ABB RAPID module: Module1.mod

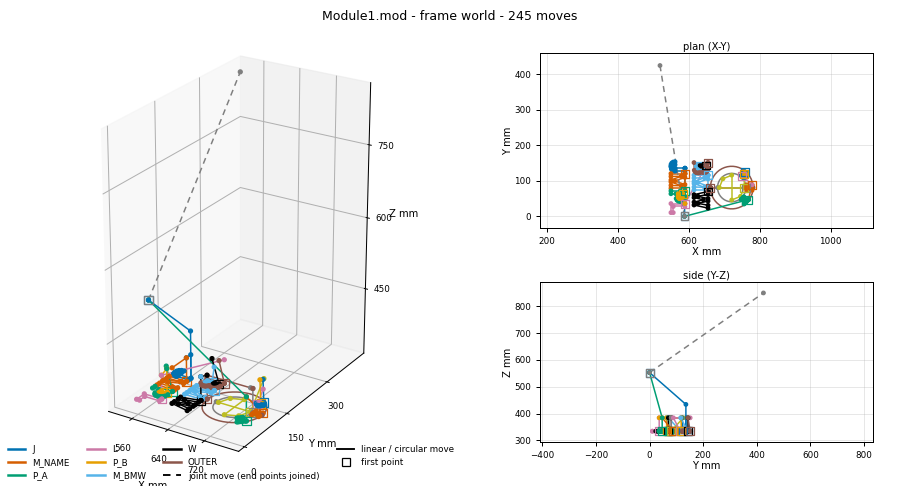
[picture p0: tool path of Module1.mod in frame world, 245 of 245 moves have a stored position in this frame; points joined in program order, loops and branches not executed]
MODULE Module1
    TASK PERS tooldata TCP_JMPL:=[TRUE,[[0,0,0],[1,0,0,0]],[1,[0,0,1],[1,0,0,0],0,0,0]];
    TASK PERS wobjdata WOB_LAB1:=[FALSE,TRUE,"",[[787.383,-61.438566881,334.26555336],[0.707106781,0,0,0.707106781]],[[0,0,0],[1,0,0,0]]];
    CONST robtarget J_10:=[[197.01,198.002626654,0.000000056],[-0.000000001,0.707106782,0.707106781,0],[0,0,0,0],[9E+09,9E+09,9E+09,9E+09,9E+09,9E+09]];
    CONST robtarget J_20:=[[197.01,225.346445883,0.000000064],[-0.000000001,0.707106782,0.707106781,0],[0,0,0,0],[9E+09,9E+09,9E+09,9E+09,9E+09,9E+09]];
    CONST robtarget J_30:=[[198.394,229.904456194,0.000000065],[-0.000000001,0.707106782,0.707106781,0],[0,0,0,0],[9E+09,9E+09,9E+09,9E+09,9E+09,9E+09]];
    CONST robtarget J_40:=[[202.114,231.501103306,0.000000066],[-0.000000001,0.707106782,0.707106781,0],[0,0,0,0],[9E+09,9E+09,9E+09,9E+09,9E+09,9E+09]];
    CONST robtarget J_50:=[[205.964,230.120830869,0.000000065],[-0.000000001,0.707106782,0.707106781,0],[0,0,0,0],[9E+09,9E+09,9E+09,9E+09,9E+09,9E+09]];
    CONST robtarget J_60:=[[206.878,228.358720771,0.000000065],[-0.000000001,0.707106782,0.707106781,0],[0,0,0,0],[9E+09,9E+09,9E+09,9E+09,9E+09,9E+09]];
    CONST robtarget J_70:=[[207.183,225.832935348,0.000000064],[-0.000000001,0.707106782,0.707106781,0],[0,0,0,0],[9E+09,9E+09,9E+09,9E+09,9E+09,9E+09]];
    CONST robtarget J_80:=[[215.378,225.832935348,0.000000064],[-0.000000001,0.707106782,0.707106781,0],[0,0,0,0],[9E+09,9E+09,9E+09,9E+09,9E+09,9E+09]];
    CONST robtarget J_90:=[[214.503,231.006128559,0.000000065],[-0.000000001,0.707106782,0.707106781,0],[0,0,0,0],[9E+09,9E+09,9E+09,9E+09,9E+09,9E+09]];
    CONST robtarget J_100:=[[211.879,234.85703209,0.000000067],[-0.000000001,0.707106782,0.707106781,0],[0,0,0,0],[9E+09,9E+09,9E+09,9E+09,9E+09,9E+09]];
    CONST robtarget J_110:=[[207.689,237.248467224,0.000000067],[-0.000000001,0.707106782,0.707106781,0],[0,0,0,0],[9E+09,9E+09,9E+09,9E+09,9E+09,9E+09]];
    CONST robtarget J_120:=[[202.114,238.046083673,0.000000067],[-0.000000001,0.707106782,0.707106781,0],[0,0,0,0],[9E+09,9E+09,9E+09,9E+09,9E+09,9E+09]];
    CONST robtarget J_130:=[[195.247,236.470649764,0.000000067],[-0.000000001,0.707106782,0.707106781,0],[0,0,0,0],[9E+09,9E+09,9E+09,9E+09,9E+09,9E+09]];
    CONST robtarget J_140:=[[192.552,234.567118309,0.000000066],[-0.000000001,0.707106782,0.707106781,0],[0,0,0,0],[9E+09,9E+09,9E+09,9E+09,9E+09,9E+09]];
    CONST robtarget J_150:=[[189.293,228.894707711,0.000000065],[-0.000000001,0.707106782,0.707106781,0],[0,0,0,0],[9E+09,9E+09,9E+09,9E+09,9E+09,9E+09]];
    CONST robtarget J_160:=[[188.876,225.346445883,0.000000064],[-0.000000001,0.707106782,0.707106781,0],[0,0,0,0],[9E+09,9E+09,9E+09,9E+09,9E+09,9E+09]];
    CONST robtarget J_170:=[[188.876,198.002626654,0.000000056],[-0.000000001,0.707106782,0.707106781,0],[0,0,0,0],[9E+09,9E+09,9E+09,9E+09,9E+09,9E+09]];
    CONST robtarget J_180:=[[197.01,198.002626654,0.000000056],[-0.000000001,0.707106782,0.707106781,0],[0,0,0,0],[9E+09,9E+09,9E+09,9E+09,9E+09,9E+09]];
    CONST robtarget M_NAME_10:=[[181.905,198.002626654,0.000000056],[-0.000000001,0.707106782,0.707106781,0],[0,0,0,0],[9E+09,9E+09,9E+09,9E+09,9E+09,9E+09]];
    CONST robtarget M_NAME_20:=[[181.905,237.500197238,0.000000067],[-0.000000001,0.707106782,0.707106781,0],[0,0,0,0],[9E+09,9E+09,9E+09,9E+09,9E+09,9E+09]];
    CONST robtarget M_NAME_30:=[[173.763,237.500197238,0.000000067],[-0.000000001,0.707106782,0.707106781,0],[0,0,0,0],[9E+09,9E+09,9E+09,9E+09,9E+09,9E+09]];
    CONST robtarget M_NAME_40:=[[174.579,208.090211995,0.000000059],[-0.000000001,0.707106782,0.707106781,0],[0,0,0,0],[9E+09,9E+09,9E+09,9E+09,9E+09,9E+09]];
    CONST robtarget M_NAME_50:=[[163.945,237.500197238,0.000000067],[-0.000000001,0.707106782,0.707106781,0],[0,0,0,0],[9E+09,9E+09,9E+09,9E+09,9E+09,9E+09]];
    CONST robtarget M_NAME_60:=[[158.355,237.500197238,0.000000067],[-0.000000001,0.707106782,0.707106781,0],[0,0,0,0],[9E+09,9E+09,9E+09,9E+09,9E+09,9E+09]];
    CONST robtarget M_NAME_70:=[[147.695,208.063341937,0.000000059],[-0.000000001,0.707106782,0.707106781,0],[0,0,0,0],[9E+09,9E+09,9E+09,9E+09,9E+09,9E+09]];
    CONST robtarget M_NAME_80:=[[148.511,237.500197238,0.000000067],[-0.000000001,0.707106782,0.707106781,0],[0,0,0,0],[9E+09,9E+09,9E+09,9E+09,9E+09,9E+09]];
    CONST robtarget M_NAME_90:=[[140.343,237.500197238,0.000000067],[-0.000000001,0.707106782,0.707106781,0],[0,0,0,0],[9E+09,9E+09,9E+09,9E+09,9E+09,9E+09]];
    CONST robtarget M_NAME_100:=[[140.343,198.002626654,0.000000056],[-0.000000001,0.707106782,0.707106781,0],[0,0,0,0],[9E+09,9E+09,9E+09,9E+09,9E+09,9E+09]];
    CONST robtarget M_NAME_110:=[[151.029,198.002626654,0.000000056],[-0.000000001,0.707106782,0.707106781,0],[0,0,0,0],[9E+09,9E+09,9E+09,9E+09,9E+09,9E+09]];
    CONST robtarget M_NAME_120:=[[161.124,226.648936574,0.000000064],[-0.000000001,0.707106782,0.707106781,0],[0,0,0,0],[9E+09,9E+09,9E+09,9E+09,9E+09,9E+09]];
    CONST robtarget M_NAME_130:=[[171.272,198.002626654,0.000000056],[-0.000000001,0.707106782,0.707106781,0],[0,0,0,0],[9E+09,9E+09,9E+09,9E+09,9E+09,9E+09]];
    CONST robtarget M_NAME_140:=[[181.905,198.002626654,0.000000056],[-0.000000001,0.707106782,0.707106781,0],[0,0,0,0],[9E+09,9E+09,9E+09,9E+09,9E+09,9E+09]];
    CONST robtarget P_A_10:=[[133.242,198.002626654,0.000000056],[-0.000000001,0.707106782,0.707106781,0],[0,0,0,0],[9E+09,9E+09,9E+09,9E+09,9E+09,9E+09]];
    CONST robtarget P_A_20:=[[133.242,237.500197238,0.000000067],[-0.000000001,0.707106782,0.707106781,0],[0,0,0,0],[9E+09,9E+09,9E+09,9E+09,9E+09,9E+09]];
    CONST robtarget P_A_30:=[[125.1,237.500197238,0.000000067],[-0.000000001,0.707106782,0.707106781,0],[0,0,0,0],[9E+09,9E+09,9E+09,9E+09,9E+09,9E+09]];
    CONST robtarget P_A_40:=[[125.1,223.584335784,0.000000063],[-0.000000001,0.707106782,0.707106781,0],[0,0,0,0],[9E+09,9E+09,9E+09,9E+09,9E+09,9E+09]];
    CONST robtarget P_A_50:=[[111.704,222.747121355,0.000000063],[-0.000000001,0.707106782,0.707106781,0],[0,0,0,0],[9E+09,9E+09,9E+09,9E+09,9E+09,9E+09]];
    CONST robtarget P_A_60:=[[106.966,220.234063855,0.000000062],[-0.000000001,0.707106782,0.707106781,0],[0,0,0,0],[9E+09,9E+09,9E+09,9E+09,9E+09,9E+09]];
    CONST robtarget P_A_70:=[[103.984,216.268609026,0.000000061],[-0.000000001,0.707106782,0.707106781,0],[0,0,0,0],[9E+09,9E+09,9E+09,9E+09,9E+09,9E+09]];
    CONST robtarget P_A_80:=[[102.99,211.075616825,0.00000006],[-0.000000001,0.707106782,0.707106781,0],[0,0,0,0],[9E+09,9E+09,9E+09,9E+09,9E+09,9E+09]];
    CONST robtarget P_A_90:=[[103.445,207.462301173,0.000000059],[-0.000000001,0.707106782,0.707106781,0],[0,0,0,0],[9E+09,9E+09,9E+09,9E+09,9E+09,9E+09]];
    CONST robtarget P_A_100:=[[104.809,204.257693241,0.000000058],[-0.000000001,0.707106782,0.707106781,0],[0,0,0,0],[9E+09,9E+09,9E+09,9E+09,9E+09,9E+09]];
    CONST robtarget P_A_110:=[[107.017,201.601800171,0.000000057],[-0.000000001,0.707106782,0.707106781,0],[0,0,0,0],[9E+09,9E+09,9E+09,9E+09,9E+09,9E+09]];
    CONST robtarget P_A_120:=[[110.004,199.630386465,0.000000057],[-0.000000001,0.707106782,0.707106781,0],[0,0,0,0],[9E+09,9E+09,9E+09,9E+09,9E+09,9E+09]];
    CONST robtarget P_A_130:=[[117.834,198.002626654,0.000000056],[-0.000000001,0.707106782,0.707106781,0],[0,0,0,0],[9E+09,9E+09,9E+09,9E+09,9E+09,9E+09]];
    CONST robtarget P_A_140:=[[133.242,198.002626654,0.000000056],[-0.000000001,0.707106782,0.707106781,0],[0,0,0,0],[9E+09,9E+09,9E+09,9E+09,9E+09,9E+09]];
    CONST robtarget L_10:=[[97.409,198.002626654,0.000000056],[-0.000000001,0.707106782,0.707106781,0],[0,-2,1,0],[9E+09,9E+09,9E+09,9E+09,9E+09,9E+09]];
    CONST robtarget L_20:=[[97.409,237.500197238,0.000000067],[-0.000000001,0.707106782,0.707106781,0],[0,-2,1,0],[9E+09,9E+09,9E+09,9E+09,9E+09,9E+09]];
    CONST robtarget L_30:=[[71.992,237.500197238,0.000000067],[-0.000000001,0.707106782,0.707106781,0],[0,-2,1,0],[9E+09,9E+09,9E+09,9E+09,9E+09,9E+09]];
    CONST robtarget L_40:=[[71.992,230.963702153,0.000000065],[-0.000000001,0.707106782,0.707106781,0],[0,-2,1,0],[9E+09,9E+09,9E+09,9E+09,9E+09,9E+09]];
    CONST robtarget L_50:=[[89.266,230.963702153,0.000000065],[-0.000000001,0.707106782,0.707106781,0],[0,-2,1,0],[9E+09,9E+09,9E+09,9E+09,9E+09,9E+09]];
    CONST robtarget L_60:=[[89.266,198.002626654,0.000000056],[-0.000000001,0.707106782,0.707106781,0],[0,-2,1,0],[9E+09,9E+09,9E+09,9E+09,9E+09,9E+09]];
    CONST robtarget L_70:=[[97.409,198.002626654,0.000000056],[-0.000000001,0.707106782,0.707106781,0],[0,-2,1,0],[9E+09,9E+09,9E+09,9E+09,9E+09,9E+09]];
    CONST robtarget P_B_100:=[[125.1,204.591447641,0.000000058],[-0.000000001,0.707106782,0.707106781,0],[0,0,0,0],[9E+09,9E+09,9E+09,9E+09,9E+09,9E+09]];
    CONST robtarget P_B_10:=[[125.1,204.591447641,0.000000058],[-0.000000001,0.707106782,0.707106781,0],[0,0,0,0],[9E+09,9E+09,9E+09,9E+09,9E+09,9E+09]];
    CONST robtarget P_B_20:=[[125.1,216.987029516,0.000000061],[-0.000000001,0.707106782,0.707106781,0],[0,0,0,0],[9E+09,9E+09,9E+09,9E+09,9E+09,9E+09]];
    CONST robtarget P_B_30:=[[117.834,216.987029516,0.000000061],[-0.000000001,0.707106782,0.707106781,0],[0,0,0,0],[9E+09,9E+09,9E+09,9E+09,9E+09,9E+09]];
    CONST robtarget P_B_40:=[[114.988,216.608020281,0.000000061],[-0.000000001,0.707106782,0.707106781,0],[0,0,0,0],[9E+09,9E+09,9E+09,9E+09,9E+09,9E+09]];
    CONST robtarget P_B_50:=[[112.908,215.46816415,0.000000061],[-0.000000001,0.707106782,0.707106781,0],[0,0,0,0],[9E+09,9E+09,9E+09,9E+09,9E+09,9E+09]];
    CONST robtarget P_B_60:=[[111.635,213.624029664,0.000000061],[-0.000000001,0.707106782,0.707106781,0],[0,0,0,0],[9E+09,9E+09,9E+09,9E+09,9E+09,9E+09]];
    CONST robtarget P_B_70:=[[111.211,211.127942727,0.00000006],[-0.000000001,0.707106782,0.707106781,0],[0,0,0,0],[9E+09,9E+09,9E+09,9E+09,9E+09,9E+09]];
    CONST robtarget P_B_80:=[[111.638,208.505990782,0.000000059],[-0.000000001,0.707106782,0.707106781,0],[0,0,0,0],[9E+09,9E+09,9E+09,9E+09,9E+09,9E+09]];
    CONST robtarget P_B_90:=[[114.957,205.083593961,0.000000058],[-0.000000001,0.707106782,0.707106781,0],[0,0,0,0],[9E+09,9E+09,9E+09,9E+09,9E+09,9E+09]];
    CONST robtarget P_B_110:=[[125.1,204.591447641,0.000000058],[-0.000000001,0.707106782,0.707106781,0],[0,0,0,0],[9E+09,9E+09,9E+09,9E+09,9E+09,9E+09]];
    CONST robtarget M_NAME_140_2:=[[177.487,133.0025429,0.000000038],[-0.000000001,0.707106782,0.707106781,0],[0,0,0,0],[9E+09,9E+09,9E+09,9E+09,9E+09,9E+09]];
    CONST robtarget M_NAME_10_2:=[[177.487,133.0025429,0.000000038],[-0.000000001,0.707106782,0.707106781,0],[0,0,0,0],[9E+09,9E+09,9E+09,9E+09,9E+09,9E+09]];
    CONST robtarget M_NAME_20_2:=[[177.487,172.500113484,0.000000049],[-0.000000001,0.707106782,0.707106781,0],[0,0,0,0],[9E+09,9E+09,9E+09,9E+09,9E+09,9E+09]];
    CONST robtarget M_NAME_30_2:=[[169.345,172.500113484,0.000000049],[-0.000000001,0.707106782,0.707106781,0],[0,0,0,0],[9E+09,9E+09,9E+09,9E+09,9E+09,9E+09]];
    CONST robtarget M_NAME_40_2:=[[170.161,143.090128241,0.000000041],[-0.000000001,0.707106782,0.707106781,0],[0,0,0,0],[9E+09,9E+09,9E+09,9E+09,9E+09,9E+09]];
    CONST robtarget M_NAME_50_2:=[[159.527,172.500113484,0.000000049],[-0.000000001,0.707106782,0.707106781,0],[0,0,0,0],[9E+09,9E+09,9E+09,9E+09,9E+09,9E+09]];
    CONST robtarget M_NAME_60_2:=[[153.937,172.500113484,0.000000049],[-0.000000001,0.707106782,0.707106781,0],[0,0,0,0],[9E+09,9E+09,9E+09,9E+09,9E+09,9E+09]];
    CONST robtarget M_NAME_70_2:=[[143.277,143.063258183,0.000000041],[-0.000000001,0.707106782,0.707106781,0],[0,0,0,0],[9E+09,9E+09,9E+09,9E+09,9E+09,9E+09]];
    CONST robtarget M_NAME_80_2:=[[144.093,172.500113484,0.000000049],[-0.000000001,0.707106782,0.707106781,0],[0,0,0,0],[9E+09,9E+09,9E+09,9E+09,9E+09,9E+09]];
    CONST robtarget M_NAME_90_2:=[[135.925,172.500113484,0.000000049],[-0.000000001,0.707106782,0.707106781,0],[0,0,0,0],[9E+09,9E+09,9E+09,9E+09,9E+09,9E+09]];
    CONST robtarget M_NAME_100_2:=[[135.925,133.0025429,0.000000038],[-0.000000001,0.707106782,0.707106781,0],[0,0,0,0],[9E+09,9E+09,9E+09,9E+09,9E+09,9E+09]];
    CONST robtarget M_NAME_110_2:=[[146.611,133.0025429,0.000000038],[-0.000000001,0.707106782,0.707106781,0],[0,0,0,0],[9E+09,9E+09,9E+09,9E+09,9E+09,9E+09]];
    CONST robtarget M_NAME_120_2:=[[156.706,161.64885282,0.000000046],[-0.000000001,0.707106782,0.707106781,0],[0,0,0,0],[9E+09,9E+09,9E+09,9E+09,9E+09,9E+09]];
    CONST robtarget M_NAME_130_2:=[[166.854,133.0025429,0.000000038],[-0.000000001,0.707106782,0.707106781,0],[0,0,0,0],[9E+09,9E+09,9E+09,9E+09,9E+09,9E+09]];
    CONST robtarget W_140:=[[131.402,133.002542901,0.000000038],[-0.000000001,0.707106782,0.707106781,0],[0,0,0,0],[9E+09,9E+09,9E+09,9E+09,9E+09,9E+09]];
    CONST robtarget W_10:=[[131.402,133.002542901,0.000000038],[-0.000000001,0.707106782,0.707106781,0],[0,0,0,0],[9E+09,9E+09,9E+09,9E+09,9E+09,9E+09]];
    CONST robtarget W_20:=[[122.635,172.500113484,0.000000049],[-0.000000001,0.707106782,0.707106781,0],[0,0,0,0],[9E+09,9E+09,9E+09,9E+09,9E+09,9E+09]];
    CONST robtarget W_30:=[[114.44,172.500113484,0.000000049],[-0.000000001,0.707106782,0.707106781,0],[0,0,0,0],[9E+09,9E+09,9E+09,9E+09,9E+09,9E+09]];
    CONST robtarget W_40:=[[108.016,146.075533071,0.000000041],[-0.000000001,0.707106782,0.707106781,0],[0,0,0,0],[9E+09,9E+09,9E+09,9E+09,9E+09,9E+09]];
    CONST robtarget W_50:=[[101.584,172.500113484,0.000000049],[-0.000000001,0.707106782,0.707106781,0],[0,0,0,0],[9E+09,9E+09,9E+09,9E+09,9E+09,9E+09]];
    CONST robtarget W_60:=[[93.39,172.500113484,0.000000049],[-0.000000001,0.707106782,0.707106781,0],[0,0,0,0],[9E+09,9E+09,9E+09,9E+09,9E+09,9E+09]];
    CONST robtarget W_70:=[[84.631,133.002542901,0.000000038],[-0.000000001,0.707106782,0.707106781,0],[0,0,0,0],[9E+09,9E+09,9E+09,9E+09,9E+09,9E+09]];
    CONST robtarget W_80:=[[92.739,133.002542901,0.000000038],[-0.000000001,0.707106782,0.707106781,0],[0,0,0,0],[9E+09,9E+09,9E+09,9E+09,9E+09,9E+09]];
    CONST robtarget W_90:=[[98.06,161.101552171,0.000000046],[-0.000000001,0.707106782,0.707106781,0],[0,0,0,0],[9E+09,9E+09,9E+09,9E+09,9E+09,9E+09]];
    CONST robtarget W_100:=[[104.544,133.002542901,0.000000038],[-0.000000001,0.707106782,0.707106781,0],[0,0,0,0],[9E+09,9E+09,9E+09,9E+09,9E+09,9E+09]];
    CONST robtarget W_110:=[[111.437,133.002542901,0.000000038],[-0.000000001,0.707106782,0.707106781,0],[0,0,0,0],[9E+09,9E+09,9E+09,9E+09,9E+09,9E+09]];
    CONST robtarget W_120:=[[117.947,161.049226269,0.000000046],[-0.000000001,0.707106782,0.707106781,0],[0,0,0,0],[9E+09,9E+09,9E+09,9E+09,9E+09,9E+09]];
    CONST robtarget W_130:=[[123.286,133.002542901,0.000000038],[-0.000000001,0.707106782,0.707106781,0],[0,0,0,0],[9E+09,9E+09,9E+09,9E+09,9E+09,9E+09]];
    CONST robtarget W_150:=[[131.402,133.0025429,0.000000038],[-0.000000001,0.707106782,0.707106781,0],[0,0,0,0],[9E+09,9E+09,9E+09,9E+09,9E+09,9E+09]];
    CONST robtarget Target_10:=[[142.499999999,126.249579958,0.000000036],[-0.000000001,0.707106782,0.707106781,0],[0,0,0,0],[9E+09,9E+09,9E+09,9E+09,9E+09,9E+09]];
    CONST robtarget Target_20:=[[202.5,66.249579958,0.000000019],[-0.000000001,0.707106782,0.707106781,0],[0,0,0,0],[9E+09,9E+09,9E+09,9E+09,9E+09,9E+09]];
    CONST robtarget Target_30:=[[142.5,6.249579958,0.000000002],[-0.000000001,0.707106782,0.707106781,0],[0,0,0,0],[9E+09,9E+09,9E+09,9E+09,9E+09,9E+09]];
    CONST robtarget Target_40:=[[82.5,66.249579958,0.000000019],[-0.000000001,0.707106782,0.707106781,0],[0,0,0,0],[9E+09,9E+09,9E+09,9E+09,9E+09,9E+09]];
    CONST robtarget Target_50:=[[142.5,126.249579958,0.000000036],[-0.000000001,0.707106782,0.707106781,0],[0,0,0,0],[9E+09,9E+09,9E+09,9E+09,9E+09,9E+09]];
    CONST robtarget Target_60:=[[142.500000001,26.249579959,0.000000007],[-0.000000001,0.707106782,0.707106781,0],[0,0,0,0],[9E+09,9E+09,9E+09,9E+09,9E+09,9E+09]];
    CONST robtarget Target_70:=[[102.5,66.249579958,0.000000019],[-0.000000001,0.707106782,0.707106781,0],[0,0,0,0],[9E+09,9E+09,9E+09,9E+09,9E+09,9E+09]];
    CONST robtarget Target_80:=[[142.5,106.249579959,0.00000003],[-0.000000001,0.707106782,0.707106781,0],[0,0,0,0],[9E+09,9E+09,9E+09,9E+09,9E+09,9E+09]];
    CONST robtarget Target_90:=[[182.5,66.249579958,0.000000019],[-0.000000001,0.707106782,0.707106781,0],[0,0,0,0],[9E+09,9E+09,9E+09,9E+09,9E+09,9E+09]];
    CONST robtarget Target_100:=[[142.5,26.249579959,0.000000007],[-0.000000001,0.707106782,0.707106781,0],[0,0,0,0],[9E+09,9E+09,9E+09,9E+09,9E+09,9E+09]];
    CONST robtarget CRUZ_70:=[[142.5,31.249877088,0.000000009],[-0.000000001,0.707106782,0.707106781,0],[0,0,0,0],[9E+09,9E+09,9E+09,9E+09,9E+09,9E+09]];
    CONST robtarget CRUZ_10:=[[142.5,31.249877088,0.000000009],[-0.000000001,0.707106782,0.707106781,0],[0,0,0,0],[9E+09,9E+09,9E+09,9E+09,9E+09,9E+09]];
    CONST robtarget CRUZ_20:=[[142.5,101.249205785,0.000000029],[-0.000000001,0.707106782,0.707106781,0],[0,0,0,0],[9E+09,9E+09,9E+09,9E+09,9E+09,9E+09]];
    CONST robtarget CRUZ_30:=[[167.249,90.998985884,0.000000026],[-0.000000001,0.707106782,0.707106781,0],[0,0,0,0],[9E+09,9E+09,9E+09,9E+09,9E+09,9E+09]];
    CONST robtarget CRUZ_40:=[[177.5,66.250248543,0.000000019],[-0.000000001,0.707106782,0.707106781,0],[0,0,0,0],[9E+09,9E+09,9E+09,9E+09,9E+09,9E+09]];
    CONST robtarget CRUZ_50:=[[107.5,66.250248543,0.000000019],[-0.000000001,0.707106782,0.707106781,0],[0,0,0,0],[9E+09,9E+09,9E+09,9E+09,9E+09,9E+09]];
    CONST robtarget CRUZ_60:=[[117.751,41.501511201,0.000000012],[-0.000000001,0.707106782,0.707106781,0],[0,0,0,0],[9E+09,9E+09,9E+09,9E+09,9E+09,9E+09]];
    CONST robtarget B_LOGO_180:=[[175.775,28.643481492,0.000000008],[-0.000000001,0.707106782,0.707106781,0],[0,0,0,0],[9E+09,9E+09,9E+09,9E+09,9E+09,9E+09]];
    CONST robtarget B_LOGO_10:=[[175.775,28.643481492,0.000000008],[-0.000000001,0.707106782,0.707106781,0],[0,-1,0,0],[9E+09,9E+09,9E+09,9E+09,9E+09,9E+09]];
    CONST robtarget B_LOGO_20:=[[175.496,27.663431494,0.000000008],[-0.000000001,0.707106782,0.707106781,0],[0,-1,0,0],[9E+09,9E+09,9E+09,9E+09,9E+09,9E+09]];
    CONST robtarget B_LOGO_30:=[[175.868,25.754243184,0.000000007],[-0.000000001,0.707106782,0.707106781,0],[0,-1,0,0],[9E+09,9E+09,9E+09,9E+09,9E+09,9E+09]];
    CONST robtarget B_LOGO_40:=[[176.493,24.932585105,0.000000007],[-0.000000001,0.707106782,0.707106781,0],[0,-1,0,0],[9E+09,9E+09,9E+09,9E+09,9E+09,9E+09]];
    CONST robtarget B_LOGO_50:=[[177.98,23.93839297,0.000000007],[-0.000000001,0.707106782,0.707106781,0],[0,-1,0,0],[9E+09,9E+09,9E+09,9E+09,9E+09,9E+09]];
    CONST robtarget B_LOGO_60:=[[179.619,23.777172624,0.000000007],[-0.000000001,0.707106782,0.707106781,0],[0,-1,0,0],[9E+09,9E+09,9E+09,9E+09,9E+09,9E+09]];
    CONST robtarget B_LOGO_70:=[[181.381,24.444681426,0.000000007],[-0.000000001,0.707106782,0.707106781,0],[0,-1,0,0],[9E+09,9E+09,9E+09,9E+09,9E+09,9E+09]];
    CONST robtarget B_LOGO_80:=[[183.239,25.938090947,0.000000007],[-0.000000001,0.707106782,0.707106781,0],[0,-1,0,0],[9E+09,9E+09,9E+09,9E+09,9E+09,9E+09]];
    CONST robtarget B_LOGO_90:=[[186.908,29.607975142,0.000000008],[-0.000000001,0.707106782,0.707106781,0],[0,-1,0,0],[9E+09,9E+09,9E+09,9E+09,9E+09,9E+09]];
    CONST robtarget B_LOGO_100:=[[176.435,40.080226571,0.000000011],[-0.000000001,0.707106782,0.707106781,0],[0,-1,0,0],[9E+09,9E+09,9E+09,9E+09,9E+09,9E+09]];
    CONST robtarget B_LOGO_110:=[[172.363,36.008705725,0.00000001],[-0.000000001,0.707106782,0.707106781,0],[0,-1,0,0],[9E+09,9E+09,9E+09,9E+09,9E+09,9E+09]];
    CONST robtarget B_LOGO_120:=[[170.989,34.225382423,0.00000001],[-0.000000001,0.707106782,0.707106781,0],[0,-1,0,0],[9E+09,9E+09,9E+09,9E+09,9E+09,9E+09]];
    CONST robtarget B_LOGO_130:=[[170.406,32.470343392,0.000000009],[-0.000000001,0.707106782,0.707106781,0],[0,-1,0,0],[9E+09,9E+09,9E+09,9E+09,9E+09,9E+09]];
    CONST robtarget B_LOGO_140:=[[170.643,30.786015039,0.000000009],[-0.000000001,0.707106782,0.707106781,0],[0,-1,0,0],[9E+09,9E+09,9E+09,9E+09,9E+09,9E+09]];
    CONST robtarget B_LOGO_150:=[[171.73,29.216237985,0.000000008],[-0.000000001,0.707106782,0.707106781,0],[0,-1,0,0],[9E+09,9E+09,9E+09,9E+09,9E+09,9E+09]];
    CONST robtarget B_LOGO_160:=[[172.662,28.516202272,0.000000008],[-0.000000001,0.707106782,0.707106781,0],[0,-1,0,0],[9E+09,9E+09,9E+09,9E+09,9E+09,9E+09]];
    CONST robtarget B_LOGO_170:=[[173.69,28.186690512,0.000000008],[-0.000000001,0.707106782,0.707106781,0],[0,-1,0,0],[9E+09,9E+09,9E+09,9E+09,9E+09,9E+09]];
    CONST robtarget M_LOGO_10:=[[150.28,8.937829714,0.000000003],[-0.000000001,0.707106782,0.707106781,0],[0,0,0,0],[9E+09,9E+09,9E+09,9E+09,9E+09,9E+09]];
    CONST robtarget M_LOGO_20:=[[150.28,23.748888353,0.000000007],[-0.000000001,0.707106782,0.707106781,0],[0,0,0,0],[9E+09,9E+09,9E+09,9E+09,9E+09,9E+09]];
    CONST robtarget M_LOGO_30:=[[147.227,23.748888353,0.000000007],[-0.000000001,0.707106782,0.707106781,0],[0,0,0,0],[9E+09,9E+09,9E+09,9E+09,9E+09,9E+09]];
    CONST robtarget M_LOGO_40:=[[147.533,12.720850994,0.000000004],[-0.000000001,0.707106782,0.707106781,0],[0,0,0,0],[9E+09,9E+09,9E+09,9E+09,9E+09,9E+09]];
    CONST robtarget M_LOGO_50:=[[143.545,23.748888353,0.000000007],[-0.000000001,0.707106782,0.707106781,0],[0,0,0,0],[9E+09,9E+09,9E+09,9E+09,9E+09,9E+09]];
    CONST robtarget M_LOGO_60:=[[141.449,23.748888353,0.000000007],[-0.000000001,0.707106782,0.707106781,0],[0,0,0,0],[9E+09,9E+09,9E+09,9E+09,9E+09,9E+09]];
    CONST robtarget M_LOGO_70:=[[137.451,12.710951499,0.000000004],[-0.000000001,0.707106782,0.707106781,0],[0,0,0,0],[9E+09,9E+09,9E+09,9E+09,9E+09,9E+09]];
    CONST robtarget M_LOGO_80:=[[137.757,23.748888353,0.000000007],[-0.000000001,0.707106782,0.707106781,0],[0,0,0,0],[9E+09,9E+09,9E+09,9E+09,9E+09,9E+09]];
    CONST robtarget M_LOGO_90:=[[134.694,23.748888353,0.000000007],[-0.000000001,0.707106782,0.707106781,0],[0,0,0,0],[9E+09,9E+09,9E+09,9E+09,9E+09,9E+09]];
    CONST robtarget M_LOGO_100:=[[134.694,8.937829714,0.000000003],[-0.000000001,0.707106782,0.707106781,0],[0,0,0,0],[9E+09,9E+09,9E+09,9E+09,9E+09,9E+09]];
    CONST robtarget M_LOGO_110:=[[138.701,8.937829714,0.000000003],[-0.000000001,0.707106782,0.707106781,0],[0,0,0,0],[9E+09,9E+09,9E+09,9E+09,9E+09,9E+09]];
    CONST robtarget M_LOGO_120:=[[142.487,19.680195934,0.000000006],[-0.000000001,0.707106782,0.707106781,0],[0,0,0,0],[9E+09,9E+09,9E+09,9E+09,9E+09,9E+09]];
    CONST robtarget M_LOGO_130:=[[146.292,8.937829714,0.000000003],[-0.000000001,0.707106782,0.707106781,0],[0,0,0,0],[9E+09,9E+09,9E+09,9E+09,9E+09,9E+09]];
    CONST robtarget M_LOGO_140:=[[150.28,8.937829714,0.000000003],[-0.000000001,0.707106782,0.707106781,0],[0,0,0,0],[9E+09,9E+09,9E+09,9E+09,9E+09,9E+09]];
    CONST robtarget W_LOGO_10:=[[108.508,19.190878041,0.000000005],[-0.000000001,0.707106782,0.707106781,0],[0,0,0,0],[9E+09,9E+09,9E+09,9E+09,9E+09,9E+09]];
    CONST robtarget W_LOGO_20:=[[116.657,31.988096567,0.000000009],[-0.000000001,0.707106782,0.707106781,0],[0,0,0,0],[9E+09,9E+09,9E+09,9E+09,9E+09,9E+09]];
    CONST robtarget W_LOGO_30:=[[114.484,34.161742813,0.00000001],[-0.000000001,0.707106782,0.707106781,0],[0,0,0,0],[9E+09,9E+09,9E+09,9E+09,9E+09,9E+09]];
    CONST robtarget W_LOGO_40:=[[105.774,28.858441954,0.000000008],[-0.000000001,0.707106782,0.707106781,0],[0,0,0,0],[9E+09,9E+09,9E+09,9E+09,9E+09,9E+09]];
    CONST robtarget W_LOGO_50:=[[111.075,37.569997498,0.000000011],[-0.000000001,0.707106782,0.707106781,0],[0,0,0,0],[9E+09,9E+09,9E+09,9E+09,9E+09,9E+09]];
    CONST robtarget W_LOGO_60:=[[108.902,39.743643743,0.000000011],[-0.000000001,0.707106782,0.707106781,0],[0,0,0,0],[9E+09,9E+09,9E+09,9E+09,9E+09,9E+09]];
    CONST robtarget W_LOGO_70:=[[96.106,31.593530983,0.000000009],[-0.000000001,0.707106782,0.707106781,0],[0,0,0,0],[9E+09,9E+09,9E+09,9E+09,9E+09,9E+09]];
    CONST robtarget W_LOGO_80:=[[98.256,29.442512155,0.000000008],[-0.000000001,0.707106782,0.707106781,0],[0,0,0,0],[9E+09,9E+09,9E+09,9E+09,9E+09,9E+09]];
    CONST robtarget W_LOGO_90:=[[107.118,35.48261828,0.00000001],[-0.000000001,0.707106782,0.707106781,0],[0,0,0,0],[9E+09,9E+09,9E+09,9E+09,9E+09,9E+09]];
    CONST robtarget W_LOGO_100:=[[101.387,26.312857542,0.000000007],[-0.000000001,0.707106782,0.707106781,0],[0,0,0,0],[9E+09,9E+09,9E+09,9E+09,9E+09,9E+09]];
    CONST robtarget W_LOGO_110:=[[103.214,24.484279405,0.000000007],[-0.000000001,0.707106782,0.707106781,0],[0,0,0,0],[9E+09,9E+09,9E+09,9E+09,9E+09,9E+09]];
    CONST robtarget W_LOGO_120:=[[112.378,30.196287984,0.000000009],[-0.000000001,0.707106782,0.707106781,0],[0,0,0,0],[9E+09,9E+09,9E+09,9E+09,9E+09,9E+09]];
    CONST robtarget W_LOGO_130:=[[106.356,21.343311083,0.000000006],[-0.000000001,0.707106782,0.707106781,0],[0,0,0,0],[9E+09,9E+09,9E+09,9E+09,9E+09,9E+09]];
    CONST robtarget W_LOGO_140:=[[108.508,19.190878041,0.000000005],[-0.000000001,0.707106782,0.707106781,0],[0,0,0,0],[9E+09,9E+09,9E+09,9E+09,9E+09,9E+09]];
    CONST robtarget B_ALOGO_10:=[[176.009,36.188310848,0.00000001],[-0.000000001,0.707106782,0.707106781,0],[0,0,0,0],[9E+09,9E+09,9E+09,9E+09,9E+09,9E+09]];
    CONST robtarget B_ALOGO_20:=[[174.161,34.339933722,0.00000001],[-0.000000001,0.707106782,0.707106781,0],[0,0,0,0],[9E+09,9E+09,9E+09,9E+09,9E+09,9E+09]];
    CONST robtarget B_ALOGO_30:=[[173.573,33.570601544,0.00000001],[-0.000000001,0.707106782,0.707106781,0],[0,0,0,0],[9E+09,9E+09,9E+09,9E+09,9E+09,9E+09]];
    CONST robtarget B_ALOGO_40:=[[173.335,32.785713016,0.000000009],[-0.000000001,0.707106782,0.707106781,0],[0,0,0,0],[9E+09,9E+09,9E+09,9E+09,9E+09,9E+09]];
    CONST robtarget B_ALOGO_50:=[[173.446,32.031937188,0.000000009],[-0.000000001,0.707106782,0.707106781,0],[0,0,0,0],[9E+09,9E+09,9E+09,9E+09,9E+09,9E+09]];
    CONST robtarget B_ALOGO_60:=[[173.91,31.354528891,0.000000009],[-0.000000001,0.707106782,0.707106781,0],[0,0,0,0],[9E+09,9E+09,9E+09,9E+09,9E+09,9E+09]];
    CONST robtarget B_ALOGO_70:=[[175.367,30.64317947,0.000000009],[-0.000000001,0.707106782,0.707106781,0],[0,0,0,0],[9E+09,9E+09,9E+09,9E+09,9E+09,9E+09]];
    CONST robtarget B_ALOGO_80:=[[176.859,31.384227376,0.000000009],[-0.000000001,0.707106782,0.707106781,0],[0,0,0,0],[9E+09,9E+09,9E+09,9E+09,9E+09,9E+09]];
    CONST robtarget B_ALOGO_90:=[[178.836,33.361297936,0.000000009],[-0.000000001,0.707106782,0.707106781,0],[0,0,0,0],[9E+09,9E+09,9E+09,9E+09,9E+09,9E+09]];
    CONST robtarget B_ALOGO_100:=[[176.009,36.188310848,0.00000001],[-0.000000001,0.707106782,0.707106781,0],[0,0,0,0],[9E+09,9E+09,9E+09,9E+09,9E+09,9E+09]];
    CONST robtarget B_ALOGO_10_2:=[[180.175,32.022037693,0.000000009],[-0.000000001,0.707106782,0.707106781,0],[0,0,0,0],[9E+09,9E+09,9E+09,9E+09,9E+09,9E+09]];
    CONST robtarget B_ALOGO_20_2:=[[178.327,30.173660567,0.000000009],[-0.000000001,0.707106782,0.707106781,0],[0,0,0,0],[9E+09,9E+09,9E+09,9E+09,9E+09,9E+09]];
    CONST robtarget B_ALOGO_30_2:=[[177.739,29.404328389,0.000000009],[-0.000000001,0.707106782,0.707106781,0],[0,0,0,0],[9E+09,9E+09,9E+09,9E+09,9E+09,9E+09]];
    CONST robtarget B_ALOGO_40_2:=[[177.501,28.619439861,0.000000008],[-0.000000001,0.707106782,0.707106781,0],[0,0,0,0],[9E+09,9E+09,9E+09,9E+09,9E+09,9E+09]];
    CONST robtarget B_ALOGO_50_2:=[[177.612,27.865664033,0.000000008],[-0.000000001,0.707106782,0.707106781,0],[0,0,0,0],[9E+09,9E+09,9E+09,9E+09,9E+09,9E+09]];
    CONST robtarget B_ALOGO_60_2:=[[178.076,27.188255736,0.000000008],[-0.000000001,0.707106782,0.707106781,0],[0,0,0,0],[9E+09,9E+09,9E+09,9E+09,9E+09,9E+09]];
    CONST robtarget B_ALOGO_70_2:=[[179.533,26.476906315,0.000000008],[-0.000000001,0.707106782,0.707106781,0],[0,0,0,0],[9E+09,9E+09,9E+09,9E+09,9E+09,9E+09]];
    CONST robtarget B_ALOGO_80_2:=[[181.025,27.217954221,0.000000008],[-0.000000001,0.707106782,0.707106781,0],[0,0,0,0],[9E+09,9E+09,9E+09,9E+09,9E+09,9E+09]];
    CONST robtarget B_ALOGO_90_2:=[[183.002,29.195024781,0.000000008],[-0.000000001,0.707106782,0.707106781,0],[0,0,0,0],[9E+09,9E+09,9E+09,9E+09,9E+09,9E+09]];
    CONST robtarget B_ALOGO_100_2:=[[180.175,32.022037693,0.000000009],[-0.000000001,0.707106782,0.707106781,0],[0,0,0,0],[9E+09,9E+09,9E+09,9E+09,9E+09,9E+09]];
    PERS tooldata MyNewTool:=[TRUE,[[68.633,0,134.238],[0.866025404,0,0.5,0]],[1,[0,0,1],[1,0,0,0],0,0,0]];
    CONST robtarget BB_BMW_10:=[[204.795566881,165.964,0.00044664],[0,0.707106781,0.707106781,0],[0,0,0,0],[9E+09,9E+09,9E+09,9E+09,9E+09,9E+09]];
    CONST robtarget BB_BMW_20:=[[197.825566881,165.964,0.00044664],[0,0.707106781,0.707106781,0],[0,0,0,0],[9E+09,9E+09,9E+09,9E+09,9E+09,9E+09]];
    CONST robtarget BB_BMW_30:=[[195.266566881,165.621,0.00044664],[0,0.707106781,0.707106781,0],[0,0,0,0],[9E+09,9E+09,9E+09,9E+09,9E+09,9E+09]];
    CONST robtarget BB_BMW_40:=[[193.337566881,164.592,0.00044664],[0,0.707106781,0.707106781,0],[0,0,0,0],[9E+09,9E+09,9E+09,9E+09,9E+09,9E+09]];
    CONST robtarget BB_BMW_50:=[[192.126566881,162.96,0.00044664],[0,0.707106781,0.707106781,0],[0,0,0,0],[9E+09,9E+09,9E+09,9E+09,9E+09,9E+09]];
    CONST robtarget BB_BMW_60:=[[191.723566881,160.807,0.00044664],[0,0.707106781,0.707106781,0],[0,0,0,0],[9E+09,9E+09,9E+09,9E+09,9E+09,9E+09]];
    CONST robtarget BB_BMW_70:=[[193.127566881,156.719,0.00044664],[0,0.707106781,0.707106781,0],[0,0,0,0],[9E+09,9E+09,9E+09,9E+09,9E+09,9E+09]];
    CONST robtarget BB_BMW_80:=[[197.339566881,155.304,0.00044664],[0,0.707106781,0.707106781,0],[0,0,0,0],[9E+09,9E+09,9E+09,9E+09,9E+09,9E+09]];
    CONST robtarget BB_BMW_90:=[[204.795566881,155.304,0.00044664],[0,0.707106781,0.707106781,0],[0,0,0,0],[9E+09,9E+09,9E+09,9E+09,9E+09,9E+09]];
    CONST robtarget BB_BMW_10_2:=[[697.791,143.357,334.266],[1,0,0,0],[0,0,0,0],[9E+09,9E+09,9E+09,9E+09,9E+09,9E+09]];
    CONST robtarget BB_BMW_20_2:=[[687.131,143.357,334.266],[1,0,0,0],[0,0,0,0],[9E+09,9E+09,9E+09,9E+09,9E+09,9E+09]];
    CONST robtarget BB_BMW_30_2:=[[687.474,133.828,334.266],[1,0,0,0],[0,0,0,0],[9E+09,9E+09,9E+09,9E+09,9E+09,9E+09]];
    CONST robtarget BB_BMW_40_2:=[[688.503,131.899,334.266],[1,0,0,0],[0,0,0,0],[9E+09,9E+09,9E+09,9E+09,9E+09,9E+09]];
    CONST robtarget BB_BMW_50_2:=[[690.135,130.688,334.266],[1,0,0,0],[0,0,0,0],[9E+09,9E+09,9E+09,9E+09,9E+09,9E+09]];
    CONST robtarget BB_BMW_60_2:=[[692.288,130.285,334.266],[1,0,0,0],[0,0,0,0],[9E+09,9E+09,9E+09,9E+09,9E+09,9E+09]];
    CONST robtarget BB_BMW_70_2:=[[696.376,131.689,334.266],[1,0,0,0],[0,0,0,0],[9E+09,9E+09,9E+09,9E+09,9E+09,9E+09]];
    CONST robtarget BB_BMW_80_2:=[[697.791,135.901,334.266],[1,0,0,0],[0,0,0,0],[9E+09,9E+09,9E+09,9E+09,9E+09,9E+09]];
    CONST robtarget BB_BMW_90_2:=[[697.791,143.357,334.266],[1,0,0,0],[0,0,0,0],[9E+09,9E+09,9E+09,9E+09,9E+09,9E+09]];
    CONST robtarget B_BWM_10:=[[704.38,151.5,334.266],[1,0,0,0],[0,0,0,0],[9E+09,9E+09,9E+09,9E+09,9E+09,9E+09]];
    CONST robtarget B_BWM_20:=[[703.692,131.344,334.266],[1,0,0,0],[0,0,0,0],[9E+09,9E+09,9E+09,9E+09,9E+09,9E+09]];
    CONST robtarget B_BWM_30:=[[701.628,126.76,334.266],[1,0,0,0],[0,0,0,0],[9E+09,9E+09,9E+09,9E+09,9E+09,9E+09]];
    CONST robtarget B_BWM_40:=[[698.234,123.974,334.266],[1,0,0,0],[0,0,0,0],[9E+09,9E+09,9E+09,9E+09,9E+09,9E+09]];
    CONST robtarget B_BWM_50:=[[693.555,123.045,334.266],[1,0,0,0],[0,0,0,0],[9E+09,9E+09,9E+09,9E+09,9E+09,9E+09]];
    CONST robtarget B_BWM_60:=[[690.827,123.417,334.266],[1,0,0,0],[0,0,0,0],[9E+09,9E+09,9E+09,9E+09,9E+09,9E+09]];
    CONST robtarget B_BWM_70:=[[688.442,124.534,334.266],[1,0,0,0],[0,0,0,0],[9E+09,9E+09,9E+09,9E+09,9E+09,9E+09]];
    CONST robtarget B_BWM_80:=[[686.526,126.316,334.266],[1,0,0,0],[0,0,0,0],[9E+09,9E+09,9E+09,9E+09,9E+09,9E+09]];
    CONST robtarget B_BWM_90:=[[685.204,128.687,334.266],[1,0,0,0],[0,0,0,0],[9E+09,9E+09,9E+09,9E+09,9E+09,9E+09]];
    CONST robtarget B_BWM_100:=[[684.055,125.97,334.266],[1,0,0,0],[0,0,0,0],[9E+09,9E+09,9E+09,9E+09,9E+09,9E+09]];
    CONST robtarget B_BWM_110:=[[682.136,123.896,334.266],[1,0,0,0],[0,0,0,0],[9E+09,9E+09,9E+09,9E+09,9E+09,9E+09]];
    CONST robtarget B_BWM_120:=[[679.574,122.581,334.266],[1,0,0,0],[0,0,0,0],[9E+09,9E+09,9E+09,9E+09,9E+09,9E+09]];
    CONST robtarget B_BWM_130:=[[676.498,122.142,334.266],[1,0,0,0],[0,0,0,0],[9E+09,9E+09,9E+09,9E+09,9E+09,9E+09]];
    CONST robtarget B_BWM_140:=[[671.488,123.051,334.266],[1,0,0,0],[0,0,0,0],[9E+09,9E+09,9E+09,9E+09,9E+09,9E+09]];
    CONST robtarget B_BWM_150:=[[667.865,125.779,334.266],[1,0,0,0],[0,0,0,0],[9E+09,9E+09,9E+09,9E+09,9E+09,9E+09]];
    CONST robtarget B_BWM_160:=[[665.654,130.189,334.266],[1,0,0,0],[0,0,0,0],[9E+09,9E+09,9E+09,9E+09,9E+09,9E+09]];
    CONST robtarget B_BWM_170:=[[664.883,136.144,334.266],[1,0,0,0],[0,0,0,0],[9E+09,9E+09,9E+09,9E+09,9E+09,9E+09]];
    CONST robtarget B_BWM_180:=[[664.883,151.5,334.266],[1,0,0,0],[0,0,0,0],[9E+09,9E+09,9E+09,9E+09,9E+09,9E+09]];
    CONST robtarget B_BWM_190:=[[704.38,151.5,334.266],[1,0,0,0],[0,0,0,0],[9E+09,9E+09,9E+09,9E+09,9E+09,9E+09]];
    CONST robtarget Target_110:=[[197.009566881,198.003,50.00044664],[0,0.707106781,0.707106781,0],[0,0,0,0],[9E+09,9E+09,9E+09,9E+09,9E+09,9E+09]];
    CONST robtarget Target_120:=[[181.905566881,198.003,50.00044664],[0,0.707106781,0.707106781,0],[0,0,0,0],[9E+09,9E+09,9E+09,9E+09,9E+09,9E+09]];
    CONST robtarget Target_130:=[[181.905566881,198.003,50.00044664],[0,0.707106781,0.707106781,0],[0,0,0,0],[9E+09,9E+09,9E+09,9E+09,9E+09,9E+09]];
    CONST robtarget Target_140:=[[133.242566881,198.003,50.00044664],[0,0.707106781,0.707106781,0],[0,0,0,0],[9E+09,9E+09,9E+09,9E+09,9E+09,9E+09]];
    CONST robtarget Target_150:=[[133.242566881,211.181,50.00044664],[0,0.707106781,0.707106781,0],[0,0,0,0],[9E+09,9E+09,9E+09,9E+09,9E+09,9E+09]];
    CONST robtarget Target_160:=[[125.099566881,204.592,50.00044664],[0,0.707106781,0.707106781,0],[0,0,0,0],[9E+09,9E+09,9E+09,9E+09,9E+09,9E+09]];
    CONST robtarget Target_270:=[[97.408566881,198.003,50.00044664],[0,0.707106781,0.707106781,0],[0,-1,0,0],[9E+09,9E+09,9E+09,9E+09,9E+09,9E+09]];
    CONST robtarget Target_280:=[[212.938566881,133.003,50.00044664],[0,0.707106781,0.707106781,0],[0,-1,0,0],[9E+09,9E+09,9E+09,9E+09,9E+09,9E+09]];
    CONST robtarget Target_170:=[[125.099566881,204.592,50.00044664],[0,0.707106781,0.707106781,0],[0,0,0,0],[9E+09,9E+09,9E+09,9E+09,9E+09,9E+09]];
    CONST robtarget Target_180:=[[97.408566881,198.003,50.00044664],[0,0.707106781,0.707106781,0],[0,0,0,0],[9E+09,9E+09,9E+09,9E+09,9E+09,9E+09]];
    CONST robtarget M_BMW150:=[[177.486566881,133.003,0.00044664],[0,0.707106781,0.707106781,0],[0,0,0,0],[9E+09,9E+09,9E+09,9E+09,9E+09,9E+09]];
    CONST robtarget M_BMW160:=[[131.401566881,133.003,50.00044664],[0,0.707106781,0.707106781,0],[0,0,0,0],[9E+09,9E+09,9E+09,9E+09,9E+09,9E+09]];
    CONST robtarget M_BMW20:=[[177.487,133.0025429,0.000000038],[-0.000000001,0.707106782,0.707106781,0],[0,0,0,0],[9E+09,9E+09,9E+09,9E+09,9E+09,9E+09]];
    CONST robtarget M_BMW10:=[[177.487,133.0025429,0.000000038],[-0.000000001,0.707106782,0.707106781,0],[0,0,0,0],[9E+09,9E+09,9E+09,9E+09,9E+09,9E+09]];
    CONST robtarget M_BMW30:=[[177.487,172.500113484,0.000000049],[-0.000000001,0.707106782,0.707106781,0],[0,0,0,0],[9E+09,9E+09,9E+09,9E+09,9E+09,9E+09]];
    CONST robtarget M_BMW40:=[[169.345,172.500113484,0.000000049],[-0.000000001,0.707106782,0.707106781,0],[0,0,0,0],[9E+09,9E+09,9E+09,9E+09,9E+09,9E+09]];
    CONST robtarget M_BMW50:=[[170.161,143.090128241,0.000000041],[-0.000000001,0.707106782,0.707106781,0],[0,0,0,0],[9E+09,9E+09,9E+09,9E+09,9E+09,9E+09]];
    CONST robtarget M_BMW60:=[[159.527,172.500113484,0.000000049],[-0.000000001,0.707106782,0.707106781,0],[0,0,0,0],[9E+09,9E+09,9E+09,9E+09,9E+09,9E+09]];
    CONST robtarget M_BMW70:=[[153.937,172.500113484,0.000000049],[-0.000000001,0.707106782,0.707106781,0],[0,0,0,0],[9E+09,9E+09,9E+09,9E+09,9E+09,9E+09]];
    CONST robtarget M_BMW80:=[[143.277,143.063258183,0.000000041],[-0.000000001,0.707106782,0.707106781,0],[0,0,0,0],[9E+09,9E+09,9E+09,9E+09,9E+09,9E+09]];
    CONST robtarget M_BMW90:=[[144.093,172.500113484,0.000000049],[-0.000000001,0.707106782,0.707106781,0],[0,0,0,0],[9E+09,9E+09,9E+09,9E+09,9E+09,9E+09]];
    CONST robtarget M_BMW100:=[[135.925,172.500113484,0.000000049],[-0.000000001,0.707106782,0.707106781,0],[0,0,0,0],[9E+09,9E+09,9E+09,9E+09,9E+09,9E+09]];
    CONST robtarget M_BMW110:=[[135.925,133.0025429,0.000000038],[-0.000000001,0.707106782,0.707106781,0],[0,0,0,0],[9E+09,9E+09,9E+09,9E+09,9E+09,9E+09]];
    CONST robtarget M_BMW120:=[[146.611,133.0025429,0.000000038],[-0.000000001,0.707106782,0.707106781,0],[0,0,0,0],[9E+09,9E+09,9E+09,9E+09,9E+09,9E+09]];
    CONST robtarget M_BMW130:=[[156.706,161.64885282,0.000000046],[-0.000000001,0.707106782,0.707106781,0],[0,0,0,0],[9E+09,9E+09,9E+09,9E+09,9E+09,9E+09]];
    CONST robtarget M_BMW140:=[[166.854,133.0025429,0.000000038],[-0.000000001,0.707106782,0.707106781,0],[0,0,0,0],[9E+09,9E+09,9E+09,9E+09,9E+09,9E+09]];
    CONST robtarget Target_290:=[[131.401566881,133.003,50.00044664],[0,0.707106781,0.707106781,0],[0,0,0,0],[9E+09,9E+09,9E+09,9E+09,9E+09,9E+09]];
    CONST robtarget Target_300:=[[142.499566881,126.25,50.00044664],[0,0.707106781,0.707106781,0],[0,0,0,0],[9E+09,9E+09,9E+09,9E+09,9E+09,9E+09]];
    CONST robtarget Target_310:=[[142.499566881,126.25,50.00044664],[0,0.707106781,0.707106781,0],[0,0,0,0],[9E+09,9E+09,9E+09,9E+09,9E+09,9E+09]];
    CONST robtarget Target_320:=[[142.499566881,26.25,50.00044664],[0,0.707106781,0.707106781,0],[0,0,0,0],[9E+09,9E+09,9E+09,9E+09,9E+09,9E+09]];
    CONST robtarget OUTER10:=[[142.499999999,126.249579958,0.000000036],[-0.000000001,0.707106782,0.707106781,0],[0,0,0,0],[9E+09,9E+09,9E+09,9E+09,9E+09,9E+09]];
    CONST robtarget OUTER20:=[[202.5,66.249579958,0.000000019],[-0.000000001,0.707106782,0.707106781,0],[0,0,0,0],[9E+09,9E+09,9E+09,9E+09,9E+09,9E+09]];
    CONST robtarget OUTER30:=[[142.5,6.249579958,0.000000002],[-0.000000001,0.707106782,0.707106781,0],[0,0,0,0],[9E+09,9E+09,9E+09,9E+09,9E+09,9E+09]];
    CONST robtarget OUTER40:=[[82.5,66.249579958,0.000000019],[-0.000000001,0.707106782,0.707106781,0],[0,0,0,0],[9E+09,9E+09,9E+09,9E+09,9E+09,9E+09]];
    CONST robtarget OUTER50:=[[142.5,126.249579958,0.000000036],[-0.000000001,0.707106782,0.707106781,0],[0,0,0,0],[9E+09,9E+09,9E+09,9E+09,9E+09,9E+09]];
    CONST robtarget Target_330:=[[142.499566881,26.25,50.00044664],[0,0.707106781,0.707106781,0],[0,0,0,0],[9E+09,9E+09,9E+09,9E+09,9E+09,9E+09]];
    CONST robtarget Target_340:=[[142.499566881,31.25,50.00044664],[0,0.707106781,0.707106781,0],[0,0,0,0],[9E+09,9E+09,9E+09,9E+09,9E+09,9E+09]];
    CONST robtarget INNER10:=[[142.500000001,26.249579959,0.000000007],[-0.000000001,0.707106782,0.707106781,0],[0,0,0,0],[9E+09,9E+09,9E+09,9E+09,9E+09,9E+09]];
    CONST robtarget INNER20:=[[102.5,66.249579958,0.000000019],[-0.000000001,0.707106782,0.707106781,0],[0,0,0,0],[9E+09,9E+09,9E+09,9E+09,9E+09,9E+09]];
    CONST robtarget INNER30:=[[142.5,106.249579959,0.00000003],[-0.000000001,0.707106782,0.707106781,0],[0,0,0,0],[9E+09,9E+09,9E+09,9E+09,9E+09,9E+09]];
    CONST robtarget INNER40:=[[182.5,66.249579958,0.000000019],[-0.000000001,0.707106782,0.707106781,0],[0,0,0,0],[9E+09,9E+09,9E+09,9E+09,9E+09,9E+09]];
    CONST robtarget INNER50:=[[142.5,26.249579959,0.000000007],[-0.000000001,0.707106782,0.707106781,0],[0,0,0,0],[9E+09,9E+09,9E+09,9E+09,9E+09,9E+09]];
    CONST robtarget Target_350:=[[142.499566881,31.25,0.00044664],[0,0.707106781,0.707106781,0],[0,0,0,0],[9E+09,9E+09,9E+09,9E+09,9E+09,9E+09]];
    CONST robtarget Target_360:=[[142.499566881,31.25,0.00044664],[0,0.707106781,0.707106781,0],[0,0,0,0],[9E+09,9E+09,9E+09,9E+09,9E+09,9E+09]];
    CONST robtarget Target_370:=[[186.908566881,29.608,50.00044664],[0,0.707106781,0.707106781,0],[0,0,0,0],[9E+09,9E+09,9E+09,9E+09,9E+09,9E+09]];
    CONST robtarget Target_380:=[[183.002566881,29.196,50.00044664],[0,0.707106781,0.707106781,0],[0,-1,0,0],[9E+09,9E+09,9E+09,9E+09,9E+09,9E+09]];
    CONST robtarget Target_410:=[[108.508566881,19.191,50.00044664],[0,0.707106781,0.707106781,0],[0,-1,0,0],[9E+09,9E+09,9E+09,9E+09,9E+09,9E+09]];
    CONST robtarget Target_400:=[[150.279566881,8.939,50.00044664],[0,0.707106781,0.707106781,0],[0,-1,0,0],[9E+09,9E+09,9E+09,9E+09,9E+09,9E+09]];
    CONST robtarget Target_390:=[[178.835566881,33.362,50.00044664],[0,0.707106781,0.707106781,0],[0,-1,0,0],[9E+09,9E+09,9E+09,9E+09,9E+09,9E+09]];
    CONST robtarget B_BMW_200:=[[204.795566881,139.592,50.00044664],[0,0.707106781,0.707106781,0],[0,0,0,0],[9E+09,9E+09,9E+09,9E+09,9E+09,9E+09]];
    CONST robtarget B_BMW_60:=[[183.580566881,160.885,0.00044664],[0,0.707106781,0.707106781,0],[0,0,0,0],[9E+09,9E+09,9E+09,9E+09,9E+09,9E+09]];
    CONST robtarget B_BMW_80:=[[185.334566881,155.247,0.00044664],[0,0.707106781,0.707106781,0],[0,0,0,0],[9E+09,9E+09,9E+09,9E+09,9E+09,9E+09]];
    CONST robtarget B_BMW_70:=[[184.019566881,157.809,0.00044664],[0,0.707106781,0.707106781,0],[0,0,0,0],[9E+09,9E+09,9E+09,9E+09,9E+09,9E+09]];
    CONST robtarget B_BMW_30:=[[191.627566881,171.729,0.00044664],[0,0.707106781,0.707106781,0],[0,0,0,0],[9E+09,9E+09,9E+09,9E+09,9E+09,9E+09]];
    CONST robtarget B_BMW_20:=[[212.938566881,172.5,0.00044664],[0,0.707106781,0.707106781,0],[0,0,0,0],[9E+09,9E+09,9E+09,9E+09,9E+09,9E+09]];
    CONST robtarget B_BMW_50:=[[184.489566881,165.895,0.00044664],[0,0.707106781,0.707106781,0],[0,0,0,0],[9E+09,9E+09,9E+09,9E+09,9E+09,9E+09]];
    CONST robtarget B_BMW_10:=[[212.938566881,133.003,0.00044664],[0,0.707106781,0.707106781,0],[0,0,0,0],[9E+09,9E+09,9E+09,9E+09,9E+09,9E+09]];
    CONST robtarget B_BMW_90:=[[187.408566881,153.328,0.00044664],[0,0.707106781,0.707106781,0],[0,0,0,0],[9E+09,9E+09,9E+09,9E+09,9E+09,9E+09]];
    CONST robtarget B_BMW_40:=[[187.217566881,169.518,0.00044664],[0,0.707106781,0.707106781,0],[0,0,0,0],[9E+09,9E+09,9E+09,9E+09,9E+09,9E+09]];
    CONST robtarget B_BMW_100:=[[190.125566881,152.179,0.00044664],[0,0.707106781,0.707106781,0],[0,0,0,0],[9E+09,9E+09,9E+09,9E+09,9E+09,9E+09]];
    CONST robtarget B_BMW_110:=[[187.754566881,150.857,0.00044664],[0,0.707106781,0.707106781,0],[0,0,0,0],[9E+09,9E+09,9E+09,9E+09,9E+09,9E+09]];
    CONST robtarget B_BMW_120:=[[185.972566881,148.941,0.00044664],[0,0.707106781,0.707106781,0],[0,0,0,0],[9E+09,9E+09,9E+09,9E+09,9E+09,9E+09]];
    CONST robtarget B_BMW_130:=[[184.855566881,146.556,0.00044664],[0,0.707106781,0.707106781,0],[0,0,0,0],[9E+09,9E+09,9E+09,9E+09,9E+09,9E+09]];
    CONST robtarget B_BMW_140:=[[184.483566881,143.828,0.00044664],[0,0.707106781,0.707106781,0],[0,0,0,0],[9E+09,9E+09,9E+09,9E+09,9E+09,9E+09]];
    CONST robtarget B_BMW_150:=[[185.412566881,139.149,0.00044664],[0,0.707106781,0.707106781,0],[0,0,0,0],[9E+09,9E+09,9E+09,9E+09,9E+09,9E+09]];
    CONST robtarget B_BMW_160:=[[188.198566881,135.755,0.00044664],[0,0.707106781,0.707106781,0],[0,0,0,0],[9E+09,9E+09,9E+09,9E+09,9E+09,9E+09]];
    CONST robtarget B_BMW_170:=[[192.782566881,133.691,0.00044664],[0,0.707106781,0.707106781,0],[0,0,0,0],[9E+09,9E+09,9E+09,9E+09,9E+09,9E+09]];
    CONST robtarget B_BMW_180:=[[199.101566881,133.003,0.00044664],[0,0.707106781,0.707106781,0],[0,0,0,0],[9E+09,9E+09,9E+09,9E+09,9E+09,9E+09]];
    CONST robtarget B_BMW_190:=[[212.938566881,133.003,0.00044664],[0,0.707106781,0.707106781,0],[0,0,0,0],[9E+09,9E+09,9E+09,9E+09,9E+09,9E+09]];
    CONST robtarget BA_BMW_100:=[[204.795566881,139.592,0.00044664],[0,0.707106781,0.707106781,0],[0,0,0,0],[9E+09,9E+09,9E+09,9E+09,9E+09,9E+09]];
    CONST robtarget BA_BMW_110:=[[204.795566881,155.304,50.00044664],[0,0.707106781,0.707106781,0],[0,0,0,0],[9E+09,9E+09,9E+09,9E+09,9E+09,9E+09]];
    CONST robtarget BA_BMW_50:=[[192.617566881,144.644,0.00044664],[0,0.707106781,0.707106781,0],[0,0,0,0],[9E+09,9E+09,9E+09,9E+09,9E+09,9E+09]];
    CONST robtarget BA_BMW_20:=[[204.795566881,149.549,0.00044664],[0,0.707106781,0.707106781,0],[0,0,0,0],[9E+09,9E+09,9E+09,9E+09,9E+09,9E+09]];
    CONST robtarget BA_BMW_60:=[[193.006566881,142.331,0.00044664],[0,0.707106781,0.707106781,0],[0,0,0,0],[9E+09,9E+09,9E+09,9E+09,9E+09,9E+09]];
    CONST robtarget BA_BMW_80:=[[196.185566881,139.887,0.00044664],[0,0.707106781,0.707106781,0],[0,0,0,0],[9E+09,9E+09,9E+09,9E+09,9E+09,9E+09]];
    CONST robtarget BA_BMW_30:=[[198.771566881,149.549,0.00044664],[0,0.707106781,0.707106781,0],[0,0,0,0],[9E+09,9E+09,9E+09,9E+09,9E+09,9E+09]];
    CONST robtarget BA_BMW_40:=[[194.155566881,148.27,0.00044664],[0,0.707106781,0.707106781,0],[0,0,0,0],[9E+09,9E+09,9E+09,9E+09,9E+09,9E+09]];
    CONST robtarget BA_BMW_10:=[[204.795566881,139.592,0.00044664],[0,0.707106781,0.707106781,0],[0,0,0,0],[9E+09,9E+09,9E+09,9E+09,9E+09,9E+09]];
    CONST robtarget BA_BMW_90:=[[199.101566881,139.592,0.00044664],[0,0.707106781,0.707106781,0],[0,0,0,0],[9E+09,9E+09,9E+09,9E+09,9E+09,9E+09]];
    CONST robtarget BA_BMW_70:=[[194.175566881,140.773,0.00044664],[0,0.707106781,0.707106781,0],[0,0,0,0],[9E+09,9E+09,9E+09,9E+09,9E+09,9E+09]];
    CONST robtarget BB_BMW_100:=[[177.486566881,133.003,50.00044664],[0,0.707106781,0.707106781,0],[0,0,0,0],[9E+09,9E+09,9E+09,9E+09,9E+09,9E+09]];
    CONST robtarget Target_420:=[[108.508566881,19.191,50.00044664],[0,0.707106781,0.707106781,0],[0,0,0,0],[9E+09,9E+09,9E+09,9E+09,9E+09,9E+09]];
    CONST robtarget Target_430:=[[-113.998809444,218.972771508,361.659146365],[0.492518449,0.507371243,0.507371243,-0.492518449],[0,0,0,1],[9E+09,9E+09,9E+09,9E+09,9E+09,9E+09]];
    CONST robtarget Target_440:=[[197.009566881,198.003,100.00044664],[0,0.707106781,0.707106781,0],[0,-1,0,0],[9E+09,9E+09,9E+09,9E+09,9E+09,9E+09]];
    CONST robtarget HOME:=[[61.438566881,199.154330601,218.677525102],[0,0.707106781,0.707106781,0],[0,0,0,0],[9E+09,9E+09,9E+09,9E+09,9E+09,9E+09]];
    CONST robtarget MANTENIMIENTO:=[[486.413239387,268.33979923,515.963180314],[0.613065878,0.352349627,0.613065804,-0.35234967],[0,0,0,1],[9E+09,9E+09,9E+09,9E+09,9E+09,9E+09]];
    PROC main()
    WHILE TRUE DO
        SetDO DO_01, 0;
        SetDO DO_02, 0;
        IF DI_01 = 1 THEN
            SetDO DO_01, 1;
            J;
            M_NAME;
            P_A;
            P_B;
            L;
            B_BMW;
            BA_BMW;
            BB_BMW;
            M_BMW;
            W;
            OUTER;
            INNER;
            CRUZ;
            B_LOGO;
            BA_LOGO;
            BB_LOGO;
            M_LOGO;
            W_LOGO;
            SetDO DO_02, 0;
        ELSEIF DI_02 = 1 THEN
            SetDO DO_02, 1;
                MANT;
            SetDO DO_02,0;
        ENDIF
    ENDWHILE
    ENDPROC

    PROC J()
        MoveJ HOME,v200,fine,MyNewTool\WObj:=WOB_LAB1;
        MoveL Target_440,v200,fine,MyNewTool\WObj:=WOB_LAB1;
        MoveL J_10,v1000,z100,MyNewTool\WObj:=WOB_LAB1;
        MoveL J_20,v1000,z100,MyNewTool\WObj:=WOB_LAB1;
        MoveL J_30,v1000,z100,MyNewTool\WObj:=WOB_LAB1;
        MoveL J_40,v1000,z100,MyNewTool\WObj:=WOB_LAB1;
        MoveL J_50,v1000,z100,MyNewTool\WObj:=WOB_LAB1;
        MoveL J_60,v1000,z100,MyNewTool\WObj:=WOB_LAB1;
        MoveL J_70,v1000,z100,MyNewTool\WObj:=WOB_LAB1;
        MoveL J_80,v1000,z100,MyNewTool\WObj:=WOB_LAB1;
        MoveL J_90,v1000,z100,MyNewTool\WObj:=WOB_LAB1;
        MoveL J_100,v1000,z100,MyNewTool\WObj:=WOB_LAB1;
        MoveL J_110,v1000,z100,MyNewTool\WObj:=WOB_LAB1;
        MoveL J_120,v1000,z100,MyNewTool\WObj:=WOB_LAB1;
        MoveL J_130,v1000,z100,MyNewTool\WObj:=WOB_LAB1;
        MoveL J_140,v1000,z100,MyNewTool\WObj:=WOB_LAB1;
        MoveL J_150,v1000,z100,MyNewTool\WObj:=WOB_LAB1;
        MoveL J_160,v1000,z100,MyNewTool\WObj:=WOB_LAB1;
        MoveL J_170,v1000,z100,MyNewTool\WObj:=WOB_LAB1;
        MoveL J_180,v1000,z100,MyNewTool\WObj:=WOB_LAB1;
        MoveL Target_110,v200,fine,MyNewTool\WObj:=WOB_LAB1;
        MoveL Target_120,v200,fine,MyNewTool\WObj:=WOB_LAB1;
    ENDPROC
    PROC M_NAME()
        MoveL M_NAME_10,v200,fine,MyNewTool\WObj:=WOB_LAB1;
        MoveL M_NAME_20,v200,fine,MyNewTool\WObj:=WOB_LAB1;
        MoveL M_NAME_30,v200,fine,MyNewTool\WObj:=WOB_LAB1;
        MoveL M_NAME_40,v200,fine,MyNewTool\WObj:=WOB_LAB1;
        MoveL M_NAME_50,v200,fine,MyNewTool\WObj:=WOB_LAB1;
        MoveL M_NAME_60,v200,fine,MyNewTool\WObj:=WOB_LAB1;
        MoveL M_NAME_70,v200,fine,MyNewTool\WObj:=WOB_LAB1;
        MoveL M_NAME_80,v200,fine,MyNewTool\WObj:=WOB_LAB1;
        MoveL M_NAME_90,v200,fine,MyNewTool\WObj:=WOB_LAB1;
        MoveL M_NAME_100,v200,fine,MyNewTool\WObj:=WOB_LAB1;
        MoveL M_NAME_110,v200,fine,MyNewTool\WObj:=WOB_LAB1;
        MoveL M_NAME_120,v200,fine,MyNewTool\WObj:=WOB_LAB1;
        MoveL M_NAME_130,v200,fine,MyNewTool\WObj:=WOB_LAB1;
        MoveL M_NAME_140,v200,fine,MyNewTool\WObj:=WOB_LAB1;
        MoveL Target_130,v200,fine,MyNewTool\WObj:=WOB_LAB1;
        MoveL Target_140,v200,fine,MyNewTool\WObj:=WOB_LAB1;
    ENDPROC
    PROC P_A()
        MoveL P_A_10,v200,fine,MyNewTool\WObj:=WOB_LAB1;
        MoveL P_A_20,v200,fine,MyNewTool\WObj:=WOB_LAB1;
        MoveL P_A_30,v200,fine,MyNewTool\WObj:=WOB_LAB1;
        MoveL P_A_40,v200,fine,MyNewTool\WObj:=WOB_LAB1;
        MoveL P_A_50,v200,fine,MyNewTool\WObj:=WOB_LAB1;
        MoveL P_A_60,v200,fine,MyNewTool\WObj:=WOB_LAB1;
        MoveL P_A_70,v200,fine,MyNewTool\WObj:=WOB_LAB1;
        MoveL P_A_80,v200,fine,MyNewTool\WObj:=WOB_LAB1;
        MoveL P_A_90,v200,fine,MyNewTool\WObj:=WOB_LAB1;
        MoveL P_A_100,v200,fine,MyNewTool\WObj:=WOB_LAB1;
        MoveL P_A_110,v200,fine,MyNewTool\WObj:=WOB_LAB1;
        MoveL P_A_120,v200,fine,MyNewTool\WObj:=WOB_LAB1;
        MoveL P_A_130,v200,fine,MyNewTool\WObj:=WOB_LAB1;
        MoveL P_A_140,v200,fine,MyNewTool\WObj:=WOB_LAB1;
        MoveL Target_150,v200,fine,MyNewTool\WObj:=WOB_LAB1;
        MoveL Target_160,v200,fine,MyNewTool\WObj:=WOB_LAB1;
    ENDPROC
    PROC L()
        MoveL L_10,v200,fine,MyNewTool\WObj:=WOB_LAB1;
        MoveL L_20,v200,fine,MyNewTool\WObj:=WOB_LAB1;
        MoveL L_30,v200,fine,MyNewTool\WObj:=WOB_LAB1;
        MoveL L_40,v200,fine,MyNewTool\WObj:=WOB_LAB1;
        MoveL L_50,v200,fine,MyNewTool\WObj:=WOB_LAB1;
        MoveL L_60,v200,fine,MyNewTool\WObj:=WOB_LAB1;
        MoveL L_70,v200,fine,MyNewTool\WObj:=WOB_LAB1;
        MoveL Target_270,v200,fine,MyNewTool\WObj:=WOB_LAB1;
        MoveL Target_280,v200,fine,MyNewTool\WObj:=WOB_LAB1;
    ENDPROC
    PROC P_B()
        MoveL P_B_100,v200,fine,MyNewTool\WObj:=WOB_LAB1;
        MoveL P_B_10,v200,fine,MyNewTool\WObj:=WOB_LAB1;
        MoveL P_B_20,v200,fine,MyNewTool\WObj:=WOB_LAB1;
        MoveL P_B_30,v200,fine,MyNewTool\WObj:=WOB_LAB1;
        MoveL P_B_40,v200,fine,MyNewTool\WObj:=WOB_LAB1;
        MoveL P_B_50,v200,fine,MyNewTool\WObj:=WOB_LAB1;
        MoveL P_B_60,v200,fine,MyNewTool\WObj:=WOB_LAB1;
        MoveL P_B_70,v200,fine,MyNewTool\WObj:=WOB_LAB1;
        MoveL P_B_80,v200,fine,MyNewTool\WObj:=WOB_LAB1;
        MoveL P_B_90,v200,fine,MyNewTool\WObj:=WOB_LAB1;
        MoveL P_B_110,v200,fine,MyNewTool\WObj:=WOB_LAB1;
        MoveL Target_170,v200,fine,MyNewTool\WObj:=WOB_LAB1;
        MoveL Target_180,v200,fine,MyNewTool\WObj:=WOB_LAB1;
    ENDPROC
    PROC M_BMW()
        MoveL M_BMW10,v200,fine,MyNewTool\WObj:=WOB_LAB1;
        MoveL M_BMW20,v200,fine,MyNewTool\WObj:=WOB_LAB1;
        MoveL M_BMW30,v200,fine,MyNewTool\WObj:=WOB_LAB1;
        MoveL M_BMW40,v200,fine,MyNewTool\WObj:=WOB_LAB1;
        MoveL M_BMW50,v200,fine,MyNewTool\WObj:=WOB_LAB1;
        MoveL M_BMW60,v200,fine,MyNewTool\WObj:=WOB_LAB1;
        MoveL M_BMW70,v200,fine,MyNewTool\WObj:=WOB_LAB1;
        MoveL M_BMW80,v200,fine,MyNewTool\WObj:=WOB_LAB1;
        MoveL M_BMW90,v200,fine,MyNewTool\WObj:=WOB_LAB1;
        MoveL M_BMW100,v200,fine,MyNewTool\WObj:=WOB_LAB1;
        MoveL M_BMW110,v200,fine,MyNewTool\WObj:=WOB_LAB1;
        MoveL M_BMW120,v200,fine,MyNewTool\WObj:=WOB_LAB1;
        MoveL M_BMW130,v200,fine,MyNewTool\WObj:=WOB_LAB1;
        MoveL M_BMW140,v200,fine,MyNewTool\WObj:=WOB_LAB1;
        MoveL M_BMW150,v200,fine,MyNewTool\WObj:=WOB_LAB1;
        MoveL M_BMW160,v200,fine,MyNewTool\WObj:=WOB_LAB1;
    ENDPROC
    PROC W()
        MoveL W_140,v200,fine,MyNewTool\WObj:=WOB_LAB1;
        MoveL W_10,v200,fine,MyNewTool\WObj:=WOB_LAB1;
        MoveL W_20,v200,fine,MyNewTool\WObj:=WOB_LAB1;
        MoveL W_30,v200,fine,MyNewTool\WObj:=WOB_LAB1;
        MoveL W_40,v200,fine,MyNewTool\WObj:=WOB_LAB1;
        MoveL W_50,v200,fine,MyNewTool\WObj:=WOB_LAB1;
        MoveL W_60,v200,fine,MyNewTool\WObj:=WOB_LAB1;
        MoveL W_70,v200,fine,MyNewTool\WObj:=WOB_LAB1;
        MoveL W_80,v200,fine,MyNewTool\WObj:=WOB_LAB1;
        MoveL W_90,v200,fine,MyNewTool\WObj:=WOB_LAB1;
        MoveL W_100,v200,fine,MyNewTool\WObj:=WOB_LAB1;
        MoveL W_110,v200,fine,MyNewTool\WObj:=WOB_LAB1;
        MoveL W_120,v200,fine,MyNewTool\WObj:=WOB_LAB1;
        MoveL W_130,v200,fine,MyNewTool\WObj:=WOB_LAB1;
        MoveL W_150,v200,fine,MyNewTool\WObj:=WOB_LAB1;
        MoveL Target_290,v200,fine,MyNewTool\WObj:=WOB_LAB1;
        MoveL Target_300,v200,fine,MyNewTool\WObj:=WOB_LAB1;
    ENDPROC
    PROC OUTER()
        MoveL OUTER10,v200,fine,MyNewTool\WObj:=WOB_LAB1;
        MoveC OUTER20,OUTER30,v200,fine,MyNewTool\WObj:=WOB_LAB1;
        MoveC OUTER40,OUTER50,v200,fine,MyNewTool\WObj:=WOB_LAB1;
        MoveL Target_310,v200,fine,MyNewTool\WObj:=WOB_LAB1;
        MoveL Target_320,v200,fine,MyNewTool\WObj:=WOB_LAB1;
    ENDPROC
    PROC INNER()
        MoveL INNER10,v200,fine,MyNewTool\WObj:=WOB_LAB1;
        MoveC INNER20,INNER30,v200,fine,MyNewTool\WObj:=WOB_LAB1;
        MoveC INNER40,INNER50,v200,fine,MyNewTool\WObj:=WOB_LAB1;
        MoveL Target_330,v200,fine,MyNewTool\WObj:=WOB_LAB1;
        MoveL Target_340,v200,fine,MyNewTool\WObj:=WOB_LAB1;
    ENDPROC
    PROC CRUZ()
        MoveL CRUZ_10,v200,fine,MyNewTool\WObj:=WOB_LAB1;
        MoveL CRUZ_20,v200,fine,MyNewTool\WObj:=WOB_LAB1;
        MoveL CRUZ_30,v200,fine,MyNewTool\WObj:=WOB_LAB1;
        MoveL CRUZ_40,v200,fine,MyNewTool\WObj:=WOB_LAB1;
        MoveL CRUZ_50,v200,fine,MyNewTool\WObj:=WOB_LAB1;
        MoveL CRUZ_60,v200,fine,MyNewTool\WObj:=WOB_LAB1;
        MoveL Target_350,v200,fine,MyNewTool\WObj:=WOB_LAB1;
        MoveL Target_360,v200,fine,MyNewTool\WObj:=WOB_LAB1;
        MoveL Target_370,v200,fine,MyNewTool\WObj:=WOB_LAB1;
    ENDPROC
    PROC B_LOGO()
        MoveL B_LOGO_90,v200,fine,MyNewTool\WObj:=WOB_LAB1;
        MoveL B_LOGO_100,v200,fine,MyNewTool\WObj:=WOB_LAB1;
        MoveL B_LOGO_110,v200,fine,MyNewTool\WObj:=WOB_LAB1;
        MoveL B_LOGO_120,v200,fine,MyNewTool\WObj:=WOB_LAB1;
        MoveL B_LOGO_130,v200,fine,MyNewTool\WObj:=WOB_LAB1;
        MoveL B_LOGO_140,v200,fine,MyNewTool\WObj:=WOB_LAB1;
        MoveL B_LOGO_150,v200,fine,MyNewTool\WObj:=WOB_LAB1;
        MoveL B_LOGO_160,v200,fine,MyNewTool\WObj:=WOB_LAB1;
        MoveL B_LOGO_170,v200,fine,MyNewTool\WObj:=WOB_LAB1;
        MoveL B_LOGO_180,v200,fine,MyNewTool\WObj:=WOB_LAB1;
        MoveL B_LOGO_10,v200,fine,MyNewTool\WObj:=WOB_LAB1;
        MoveL B_LOGO_20,v200,fine,MyNewTool\WObj:=WOB_LAB1;
        MoveL B_LOGO_30,v200,fine,MyNewTool\WObj:=WOB_LAB1;
        MoveL B_LOGO_40,v200,fine,MyNewTool\WObj:=WOB_LAB1;
        MoveL B_LOGO_50,v200,fine,MyNewTool\WObj:=WOB_LAB1;
        MoveL B_LOGO_60,v200,fine,MyNewTool\WObj:=WOB_LAB1;
        MoveL B_LOGO_70,v200,fine,MyNewTool\WObj:=WOB_LAB1;
        MoveL B_LOGO_80,v200,fine,MyNewTool\WObj:=WOB_LAB1;
        MoveL B_LOGO_90,v200,fine,MyNewTool\WObj:=WOB_LAB1;
        MoveL Target_380,v200,fine,MyNewTool\WObj:=WOB_LAB1;
    ENDPROC
    PROC M_LOGO()
        MoveL M_LOGO_10,v200,fine,MyNewTool\WObj:=WOB_LAB1;
        MoveL M_LOGO_20,v200,fine,MyNewTool\WObj:=WOB_LAB1;
        MoveL M_LOGO_30,v200,fine,MyNewTool\WObj:=WOB_LAB1;
        MoveL M_LOGO_40,v200,fine,MyNewTool\WObj:=WOB_LAB1;
        MoveL M_LOGO_50,v200,fine,MyNewTool\WObj:=WOB_LAB1;
        MoveL M_LOGO_60,v200,fine,MyNewTool\WObj:=WOB_LAB1;
        MoveL M_LOGO_70,v200,fine,MyNewTool\WObj:=WOB_LAB1;
        MoveL M_LOGO_80,v200,fine,MyNewTool\WObj:=WOB_LAB1;
        MoveL M_LOGO_90,v200,fine,MyNewTool\WObj:=WOB_LAB1;
        MoveL M_LOGO_100,v200,fine,MyNewTool\WObj:=WOB_LAB1;
        MoveL M_LOGO_110,v200,fine,MyNewTool\WObj:=WOB_LAB1;
        MoveL M_LOGO_120,v200,fine,MyNewTool\WObj:=WOB_LAB1;
        MoveL M_LOGO_130,v200,fine,MyNewTool\WObj:=WOB_LAB1;
        MoveL M_LOGO_140,v200,fine,MyNewTool\WObj:=WOB_LAB1;
        MoveL Target_410,v200,fine,MyNewTool\WObj:=WOB_LAB1;
    ENDPROC
    PROC W_LOGO()
        MoveL W_LOGO_10,v200,fine,MyNewTool\WObj:=WOB_LAB1;
        MoveL W_LOGO_20,v200,fine,MyNewTool\WObj:=WOB_LAB1;
        MoveL W_LOGO_30,v200,fine,MyNewTool\WObj:=WOB_LAB1;
        MoveL W_LOGO_40,v200,fine,MyNewTool\WObj:=WOB_LAB1;
        MoveL W_LOGO_50,v200,fine,MyNewTool\WObj:=WOB_LAB1;
        MoveL W_LOGO_60,v200,fine,MyNewTool\WObj:=WOB_LAB1;
        MoveL W_LOGO_70,v200,fine,MyNewTool\WObj:=WOB_LAB1;
        MoveL W_LOGO_80,v200,fine,MyNewTool\WObj:=WOB_LAB1;
        MoveL W_LOGO_90,v200,fine,MyNewTool\WObj:=WOB_LAB1;
        MoveL W_LOGO_100,v200,fine,MyNewTool\WObj:=WOB_LAB1;
        MoveL W_LOGO_110,v200,fine,MyNewTool\WObj:=WOB_LAB1;
        MoveL W_LOGO_120,v200,fine,MyNewTool\WObj:=WOB_LAB1;
        MoveL W_LOGO_130,v200,fine,MyNewTool\WObj:=WOB_LAB1;
        MoveL W_LOGO_140,v200,fine,MyNewTool\WObj:=WOB_LAB1;
        MoveL Target_420,v200,fine,MyNewTool\WObj:=WOB_LAB1;
        MoveL HOME,v200,fine,MyNewTool\WObj:=WOB_LAB1;
    ENDPROC
    PROC BA_LOGO()
        MoveL B_ALOGO_10,v200,fine,MyNewTool\WObj:=WOB_LAB1;
        MoveL B_ALOGO_20,v200,fine,MyNewTool\WObj:=WOB_LAB1;
        MoveL B_ALOGO_30,v200,fine,MyNewTool\WObj:=WOB_LAB1;
        MoveL B_ALOGO_40,v200,fine,MyNewTool\WObj:=WOB_LAB1;
        MoveL B_ALOGO_50,v200,fine,MyNewTool\WObj:=WOB_LAB1;
        MoveL B_ALOGO_60,v200,fine,MyNewTool\WObj:=WOB_LAB1;
        MoveL B_ALOGO_70,v200,fine,MyNewTool\WObj:=WOB_LAB1;
        MoveL B_ALOGO_80,v200,fine,MyNewTool\WObj:=WOB_LAB1;
        MoveL B_ALOGO_90,v200,fine,MyNewTool\WObj:=WOB_LAB1;
        MoveL B_ALOGO_100,v200,fine,MyNewTool\WObj:=WOB_LAB1;
        MoveL Target_400,v200,fine,MyNewTool\WObj:=WOB_LAB1;
    ENDPROC
    PROC BB_LOGO()
        MoveL B_ALOGO_10_2,v200,fine,MyNewTool\WObj:=WOB_LAB1;
        MoveL B_ALOGO_20_2,v200,fine,MyNewTool\WObj:=WOB_LAB1;
        MoveL B_ALOGO_30_2,v200,fine,MyNewTool\WObj:=WOB_LAB1;
        MoveL B_ALOGO_40_2,v200,fine,MyNewTool\WObj:=WOB_LAB1;
        MoveL B_ALOGO_50_2,v200,fine,MyNewTool\WObj:=WOB_LAB1;
        MoveL B_ALOGO_60_2,v200,fine,MyNewTool\WObj:=WOB_LAB1;
        MoveL B_ALOGO_70_2,v200,fine,MyNewTool\WObj:=WOB_LAB1;
        MoveL B_ALOGO_80_2,v200,fine,MyNewTool\WObj:=WOB_LAB1;
        MoveL B_ALOGO_90_2,v200,fine,MyNewTool\WObj:=WOB_LAB1;
        MoveL B_ALOGO_100_2,v200,fine,MyNewTool\WObj:=WOB_LAB1;
        MoveL Target_390,v200,fine,MyNewTool\WObj:=WOB_LAB1;
    ENDPROC
    PROC BB_BMW()
        MoveL BB_BMW_90,v200,fine,MyNewTool\WObj:=WOB_LAB1;
        MoveL BB_BMW_10,v200,fine,MyNewTool\WObj:=WOB_LAB1;
        MoveL BB_BMW_20,v200,fine,MyNewTool\WObj:=WOB_LAB1;
        MoveL BB_BMW_30,v200,fine,MyNewTool\WObj:=WOB_LAB1;
        MoveL BB_BMW_40,v200,fine,MyNewTool\WObj:=WOB_LAB1;
        MoveL BB_BMW_50,v200,fine,MyNewTool\WObj:=WOB_LAB1;
        MoveL BB_BMW_60,v200,fine,MyNewTool\WObj:=WOB_LAB1;
        MoveL BB_BMW_70,v200,fine,MyNewTool\WObj:=WOB_LAB1;
        MoveL BB_BMW_80,v200,fine,MyNewTool\WObj:=WOB_LAB1;
        MoveL BB_BMW_90,v200,fine,MyNewTool\WObj:=WOB_LAB1;
        MoveL BB_BMW_100,v200,fine,MyNewTool\WObj:=WOB_LAB1;
    ENDPROC
    PROC BA_BMW()
        MoveL BA_BMW_10,v200,fine,MyNewTool\WObj:=WOB_LAB1;
        MoveL BA_BMW_20,v200,fine,MyNewTool\WObj:=WOB_LAB1;
        MoveL BA_BMW_30,v200,fine,MyNewTool\WObj:=WOB_LAB1;
        MoveL BA_BMW_40,v200,fine,MyNewTool\WObj:=WOB_LAB1;
        MoveL BA_BMW_50,v200,fine,MyNewTool\WObj:=WOB_LAB1;
        MoveL BA_BMW_60,v200,fine,MyNewTool\WObj:=WOB_LAB1;
        MoveL BA_BMW_70,v200,fine,MyNewTool\WObj:=WOB_LAB1;
        MoveL BA_BMW_80,v200,fine,MyNewTool\WObj:=WOB_LAB1;
        MoveL BA_BMW_90,v200,fine,MyNewTool\WObj:=WOB_LAB1;
        MoveL BA_BMW_100,v200,fine,MyNewTool\WObj:=WOB_LAB1;
        MoveL BA_BMW_110,v200,fine,MyNewTool\WObj:=WOB_LAB1;
    ENDPROC
    PROC B_BMW()
        MoveL B_BMW_10,v200,fine,MyNewTool\WObj:=WOB_LAB1;
        MoveL B_BMW_20,v200,fine,MyNewTool\WObj:=WOB_LAB1;
        MoveL B_BMW_30,v200,fine,MyNewTool\WObj:=WOB_LAB1;
        MoveL B_BMW_40,v200,fine,MyNewTool\WObj:=WOB_LAB1;
        MoveL B_BMW_50,v200,fine,MyNewTool\WObj:=WOB_LAB1;
        MoveL B_BMW_60,v200,fine,MyNewTool\WObj:=WOB_LAB1;
        MoveL B_BMW_70,v200,fine,MyNewTool\WObj:=WOB_LAB1;
        MoveL B_BMW_80,v200,fine,MyNewTool\WObj:=WOB_LAB1;
        MoveL B_BMW_90,v200,fine,MyNewTool\WObj:=WOB_LAB1;
        MoveL B_BMW_100,v200,fine,MyNewTool\WObj:=WOB_LAB1;
        MoveL B_BMW_110,v200,fine,MyNewTool\WObj:=WOB_LAB1;
        MoveL B_BMW_120,v200,fine,MyNewTool\WObj:=WOB_LAB1;
        MoveL B_BMW_130,v200,fine,MyNewTool\WObj:=WOB_LAB1;
        MoveL B_BMW_140,v200,fine,MyNewTool\WObj:=WOB_LAB1;
        MoveL B_BMW_150,v200,fine,MyNewTool\WObj:=WOB_LAB1;
        MoveL B_BMW_160,v200,fine,MyNewTool\WObj:=WOB_LAB1;
        MoveL B_BMW_170,v200,fine,MyNewTool\WObj:=WOB_LAB1;
        MoveL B_BMW_180,v200,fine,MyNewTool\WObj:=WOB_LAB1;
        MoveL B_BMW_190,v200,fine,MyNewTool\WObj:=WOB_LAB1;
        MoveL B_BMW_200,v200,fine,MyNewTool\WObj:=WOB_LAB1;
    ENDPROC
    PROC MANT()
        MoveJ HOME,v200,fine,MyNewTool\WObj:=WOB_LAB1;
        MoveJ MANTENIMIENTO,v200,fine,MyNewTool\WObj:=WOB_LAB1;
    ENDPROC
ENDMODULE
